Universal Robots PolyScope program: v2ross_dia8V2.urp

Program v2ross_dia8V2 (installation=botross directory=/programs/usbdisk/APS2OsUltimosRomanticos createdIn=3.15.3.106223 lastSavedIn=3.15.3.106223 robotSerialNumber=2017357016)
Calibrated DH parameters: a=[0.000147, -0.403633, -0.391058, 0.000042, 0.000118, 0]; d=[0.089178, 30.14366, -33.809995, 3.776935, 0.094786, 0.082481]; alpha=[1.56929, -0.004446, 0.00863, 1.569893, -1.570304, 0]; deltaTheta=[0.000049, -0.320568, 0.239888, 0.08077, 0.000061, 0.000065]
BeforeStart
  Socket_color := socket_open("10.103.16.232",30001,socket_name="color")
  Socket_coord := socket_open("10.103.16.232",30002,socket_name="coord")
  points_done := ""
  ready_to_move := False
Robot Program (runOnlyOnce=false)
  points_done := socket_read_string(socket_name="color")
  If points_done ≟ "Color is done"
    Script: socket_close(socket_name="coord")
    Socket_coord := False
  Loop While (checkContinuously=false) expression=Socket_color ≟  False
    Socket_color := socket_open("10.103.16.232",30001,socket_name="color")
  'Ready to recieve coordinates from a color'
  Loop While (checkContinuously=false) expression=Socket_coord ≟ False
    Socket_coord := socket_open("10.103.16.232",30002,socket_name="coord")
    Script: socket_send_string("ready",socket_name="color")
  Num_points := socket_read_ascii_float(1,socket_name="coord")
  N := Num_points[1]
  X := socket_read_ascii_float(N,socket_name="coord")
  Y := socket_read_ascii_float(N,socket_name="coord")
  Z := socket_read_ascii_float(N,socket_name="coord")
  count := 1
  Loop While (checkContinuously=false) expression=count≤N
    move2pose := p[X[count]/1000,Y[count]/1000,Z[count]/1000,0,0,0]
    MoveL speed 200 mm/s, acceleration 600 mm/s^2 (useActiveTCP=true) feature=Plano_Pintura
      Waypoint Waypoint (Variable): variable=move2pose
    count := count+1
  If X[10] ≟ 0  and Y[10] ≟ 0
    Script: socket_send_string("robot_operation_done",socket_name="coord")
    SuppressedNode
      Script: socket_send_string("ready",socket_name="color")
